FUNCTION_BLOCK FB_TcExternalTime
VAR
	_hr : HRESULT;
	_ipExtTime : ITcExternalTime;
	_eTimeType: ETcExternalTimeType;
END_VAR

METHOD FB_Exit : BOOL
VAR_INPUT
	bInCopyCode : BOOL; // if TRUE, the exit method is called for exiting an instance that is copied afterwards (online change).
END_VAR
IF _ipExtTime <> 0 THEN
	FW_SafeRelease(ADR(_ipExtTime));
END_IF
END_METHOD

METHOD FB_Init : BOOL
VAR_INPUT
	bInitRetains : BOOL; // if TRUE, the retain variables are initialized (warm start / cold start)
	bInCopyCode : BOOL;  // if TRUE, the instance afterwards gets moved into the copy code (online change)
	eTimeType : ETcExternalTimeType; 
END_VAR
VAR
	ipServer : ITComObjectServer;
END_VAR
ipServer := TwinCAT_SystemInfoVarList._AppInfo.TComSrvPtr;
_eTimeType := eTimeType; 
IF _ipExtTime = 0 THEN
	_hr := ipServer.TcQueryInterface(IID_ITcExternalTime, ADR(_ipExtTime));
	IF FAILED(_hr) THEN RETURN; END_IF
END_IF
END_METHOD

METHOD GetExternalOffset : LINT
VAR_INPUT
END_VAR
IF _ipExtTime <> 0 THEN
	_hr := _ipExtTime.GetExternalTimeOffset(_eTimeType, GetExternalOffset);
	IF _hr <> 0 THEN GetExternalOffset := 0; END_IF
END_IF
END_METHOD

METHOD GetExternalTime : LINT
VAR_INPUT
END_VAR
IF _ipExtTime <> 0 THEN
	GetExternalTime := GetSystemTime();
	_hr := _ipExtTime.SystemTimeToExternalTime(_eTimeType, GetExternalTime);
	IF _hr <> 0 THEN GetExternalTime := 0; END_IF
END_IF
END_METHOD

METHOD GetSystemTime : LINT
GetSystemTime := ULINT_TO_LINT(F_GetSystemTime());
END_METHOD

PROPERTY Result : HRESULT
GET
Result := _hr;
END_GET
END_PROPERTY

END_FUNCTION_BLOCK

(* stored: Version 1.1.0.1, ProductVersion 3.1.4024.9
   POU FB_TcExternalTime: Id {04df80b6-ee6b-4d8a-bf76-590aa477e691}, SpecialFunc None
   Method FB_Exit: Id {6c2b1820-259c-4133-898f-66a50195986e}
   Method FB_Init: Id {10fb0437-74a0-4795-85cb-4994f004472a}
   Method GetExternalOffset: Id {3d9bdbf0-d24c-49b2-9bec-300aff29aee6}
   Method GetExternalTime: Id {b62b48e8-3381-4463-bee1-10cde8a1c840}
   Method GetSystemTime: Id {e6892a87-bc2b-436a-a81b-d7c86e36956d}
   Property Result: Id {1113eba2-31a7-489b-a3a5-e8fc7e7f6e95}
   Get Get: Id {277aeb5d-98f6-4a35-8443-65530252d50d} *)
